INTERFACE I_XtsHardware

PROPERTY AllMoverPositionsValid : BOOL
GET
END_GET
END_PROPERTY

PROPERTY AnyPartsInError : BOOL
GET
END_GET
END_PROPERTY

METHOD AreExpectedMoversFound : BOOL
VAR_INPUT
END_VAR
END_METHOD

PROPERTY DetectedNumberOfParts : INT
GET
END_GET
END_PROPERTY

PROPERTY DetectedNumberOfTracks : UINT
GET
END_GET
END_PROPERTY

PROPERTY ExpectedNumberOfParts : int
GET
END_GET
SET
END_SET
END_PROPERTY

PROPERTY ExpectedNumberOfTracks : int
GET
END_GET
SET
END_SET
END_PROPERTY

METHOD GetConfiguredDetectionMoverNumber : UDINT
VAR_INPUT
END_VAR
END_METHOD

METHOD GetMoverDetectionState : DetectionStateEnum
VAR_INPUT
END_VAR
END_METHOD

METHOD getNumberMoversDetected : UDINT
VAR_INPUT
END_VAR
END_METHOD

METHOD GetPartErrorCode : UDINT
END_METHOD

METHOD GetTrackInterfaceByNumber : I_XtsTrack
VAR_INPUT
	TrackNumber : UINT;
END_VAR
END_METHOD

METHOD GetTrackInterfaceByOTCID : I_XtsTrack
VAR_INPUT
	trackOTCID : OTCID;
END_VAR
END_METHOD

METHOD HasValidXPUReference : BOOL
VAR_INPUT
END_VAR
END_METHOD

PROPERTY Initialised : BOOL
GET
END_GET
END_PROPERTY

METHOD IsHardware24VdcOK : HRESULT
VAR_INPUT
END_VAR
END_METHOD

METHOD IsHardware48VdcOK : HRESULT
VAR_INPUT
END_VAR
END_METHOD

METHOD IsIDDetectionStandard : BOOL
VAR_INPUT
END_VAR
END_METHOD

PROPERTY MyName : string
GET
END_GET
END_PROPERTY

PROPERTY MyXpu : I_TcIoXtsProcessingUnit
GET
END_GET
SET
END_SET
END_PROPERTY

PROPERTY MyXts : INT
GET
END_GET
SET
END_SET
END_PROPERTY

METHOD RemoveATrackFromDetection : HRESULT
VAR_INPUT
	TrackToRemove : UINT;
END_VAR
END_METHOD

METHOD ResetAllParts : BOOL
END_METHOD

METHOD ResetAPart : HRESULT
VAR_INPUT
	Part : UINT;
END_VAR
END_METHOD

METHOD SetATrackForDetection : HRESULT
VAR_INPUT
	TrackToDetect : UINT;
END_VAR
END_METHOD

METHOD SetMoverNumberForDetection : HRESULT
VAR_INPUT
	NumberOfMovers : INT;
END_VAR
END_METHOD

METHOD TriggerMoverDetection : HRESULT
VAR_INPUT
END_VAR
END_METHOD

METHOD TriggerMoverIDDetection : HRESULT
VAR_INPUT
END_VAR
END_METHOD

METHOD TriggerMoverRedetection : HRESULT
VAR_INPUT
END_VAR
END_METHOD

PROPERTY XtsInSim : BOOL
GET
END_GET
END_PROPERTY

END_INTERFACE

(* stored: Version 1.1.0.1
   Itf I_XtsHardware: Id {9afac880-0754-4de0-b157-657ea2ab2f5c}
   Folder Commands: Id {27c9da71-387e-4094-ae9a-f077ff9b1b1e}
   Folder Settings: Id {e3948c37-e7d1-40e0-b3aa-465d52d19205}
   Folder Status: Id {f56f8332-a404-49a0-b1fa-c3796e00575d}
   Property AllMoverPositionsValid: Id {e2e91fe2-3894-447f-80d4-305bc049477e}
   Get Get: Id {e30d4cf5-dc43-4863-88ad-102cf2d59f9a}
   Property AnyPartsInError: Id {422c42a2-256b-4d64-8b66-743786694e0c}
   Get Get: Id {aca19c6b-382e-43b6-92f3-3dd92a1a8736}
   Method AreExpectedMoversFound: Id {aa48d66d-e689-4a24-808d-2ead7682c5a9}
   Property DetectedNumberOfParts: Id {26f59286-1828-426d-8401-9c022372b2b3}
   Get Get: Id {be1603c2-e62c-4ec9-9bc8-45b0c3dfbaa1}
   Property DetectedNumberOfTracks: Id {1f7b777e-4e84-4e05-a960-b4258ee4a093}
   Get Get: Id {b975fd9f-07a4-422f-a5dd-e3785eb793b3}
   Property ExpectedNumberOfParts: Id {8baf703f-4030-43b9-bdf8-f6888d62a51a}
   Get Get: Id {0b7c22e3-40c5-447c-8669-8bda14b6c107}
   Set Set: Id {5fd5e677-eecf-47de-bd59-50e6a5a429b3}
   Property ExpectedNumberOfTracks: Id {060a46c5-290c-4bcd-90e6-de762c9e2c08}
   Get Get: Id {32b0bf5c-9771-495a-89d6-3032bdd0b8c3}
   Set Set: Id {9407f136-b996-42ff-9b05-517db21ec39e}
   Method GetConfiguredDetectionMoverNumber: Id {840a6c17-fbef-4810-9acd-02a47aa8f2b0}
   Method GetMoverDetectionState: Id {fa37bb06-5333-4945-837b-ed2607a0f10b}
   Method getNumberMoversDetected: Id {f24c38ad-dbfa-488d-af77-9f21cd2a2d34}
   Method GetPartErrorCode: Id {a778e153-11fc-44a4-9a30-e1a939a035d7}
   Method GetTrackInterfaceByNumber: Id {fdddf6a5-daa4-4b5f-bc28-556a31f03729}
   Method GetTrackInterfaceByOTCID: Id {32320bf3-efb9-473d-bca7-a0ced8f8657b}
   Method HasValidXPUReference: Id {4bb0c294-1f51-4661-82c9-c8d7d52811fe}
   Property Initialised: Id {f239fb15-642d-4faf-9558-f276626556b5}
   Get Get: Id {9924b9ef-90c1-4085-a436-bbc9b1c7f93e}
   Method IsHardware24VdcOK: Id {d84db133-10f1-4c84-aee2-357bd38938fd}
   Method IsHardware48VdcOK: Id {df545d44-305d-4b7a-922f-4b561f83d56a}
   Method IsIDDetectionStandard: Id {812f54c9-547b-4e7f-8855-88380dcaf23c}
   Property MyName: Id {b43d0e80-e621-46e0-af70-0a677800dc98}
   Get Get: Id {494ebcb6-a0a6-498f-a4fa-49193344e0b2}
   Property MyXpu: Id {e2e815a3-d77a-4532-829a-eddabfcaecf8}
   Get Get: Id {bcee566b-b874-4152-ba22-6584fd88703d}
   Set Set: Id {98412ca9-12f3-48a0-a17f-85457d787566}
   Property MyXts: Id {53462daf-bea5-4a22-960f-7d5bfcc2ce3c}
   Get Get: Id {0d7e989b-6c34-4c03-ad75-2a4dfad812ae}
   Set Set: Id {09a1cb2a-649a-43ca-b93f-1edc829a7cd1}
   Method RemoveATrackFromDetection: Id {6b996083-6718-40f8-8385-c5509d71f04d}
   Method ResetAllParts: Id {1ef4fc6a-84af-4fb3-a74e-14a888b66822}
   Method ResetAPart: Id {7685d8b6-69e4-4d21-b6d9-56ad03f5a9bf}
   Method SetATrackForDetection: Id {e5174e94-1d43-416d-9cf0-82b8810737fe}
   Method SetMoverNumberForDetection: Id {7821c5af-a98b-4e00-bdec-978858c91986}
   Method TriggerMoverDetection: Id {3ca79f9d-8f1a-40ef-9b71-3df667743234}
   Method TriggerMoverIDDetection: Id {94d400e7-7631-41b8-b1e4-2b7514685c32}
   Method TriggerMoverRedetection: Id {02f3159c-a37c-4b20-ae4e-7c65bf1966cb}
   Property XtsInSim: Id {e7984951-80bc-4277-8802-61a242b4487d}
   Get Get: Id {68f8f64f-28c5-45c5-818b-d199ab177846} *)
